{attribute 'qualified_only'}
VAR_GLOBAL
	Bin1Full : BOOL := TRUE;
	Bin2Full : BOOL := TRUE;
	Bin3Full : BOOL := TRUE;
	Bin4Full : BOOL := TRUE;

END_VAR

(* stored: Version 1.1.0.1, ProductVersion 3.1.4024.13
   GVL BinSensorsFromPlc2: Id {0fad800c-6356-46ac-bc47-00ce59469623} *)
